TYPE FfuConfigs :
STRUCT
	Astrofan612FfuConfig : Astrofan612FfuConfig;
END_STRUCT
END_TYPE

(* stored: Version 1.1.0.1, ProductVersion 3.1.4024.12
   DUT FfuConfigs: Id {46336bd1-9a51-4272-8675-5d184b8ca5b0} *)
